FUNCTION_BLOCK FB_HybridStarter EXTENDS FB_BaseDevice
VAR_INPUT
	// The control output to the starter
    ControlOutput    AT %Q* : UINT;
	// The 5in1 state data word from the starter
    StatusInput      AT %I* : UINT;
	// The Max. current ampere word from the starter, in 10s of mA
    CurrentMaxInput  AT %I* : UINT;
	// The Thermal load input word from the starter
    ThermalLoadInput AT %I* : UINT;

    // Local copy of main control word as UINT (same as ControlOutput)
    uControl : UINT;
    // Local copy of main control word, individual bits that are translated to send to output
    stControl : ST_HybridStarterControlOutputBits;

    // Local copy of main status word as UINT (same as StatusInput)
    uStatus : UINT;
    // Local copy of main status word, translated to be readable as individual bits
    stStatus : ST_HybridStarterControlInputBits;

    // Max current word, multiplied by 10x, from tens of mA (same as CurrentMaxInput) to hundreds of mA, to be human readable
    uCurrentMilliamps : UINT;

    // Motor thermal load percentage (same as ThermalLoadInput)
    uThermalLoadPercent : UINT;
END_VAR

VAR
    uControlOutput : U_HybridStarterControlOutput;
    uControlInput1 : U_HybridStarterControlInput;
END_VAR

METHOD ReadControlInputs : BOOL
uStatus             := StatusInput;
uCurrentMilliamps   := CurrentMaxInput * 10; // Turn the 10s of mA value into 100s of mA
uThermalLoadPercent := ThermalLoadInput;

// Run the main input UINT through the union and store the bits in the local struct VAR
uControlInput1.uUint := uStatus;
stStatus             := uControlInput1.stBits;

ReadControlInputs := TRUE;
END_METHOD

METHOD RunForward : BOOL
VAR_INPUT
END_VAR
stControl.ForwardRunning := TRUE;
stControl.ReverseRunning := FALSE;
RunForward := TRUE;
END_METHOD

METHOD RunReverse : BOOL
VAR_INPUT
END_VAR
stControl.ForwardRunning := FALSE;
stControl.ReverseRunning := TRUE;
RunReverse := TRUE;
END_METHOD

METHOD SetNominalCurrent : BOOL
VAR_INPUT
	bit0 : BOOL;
	bit1 : BOOL;
	bit2 : BOOL;
	bit3 : BOOL;
END_VAR
stControl.NominalMotorCurrent0 := bit0;
stControl.NominalMotorCurrent1 := bit1;
stControl.NominalMotorCurrent2 := bit2;
stControl.NominalMotorCurrent3 := bit3;
stControl.IdentificationValid := TRUE;
SetNominalCurrent := TRUE;
END_METHOD

METHOD Stop : BOOL
VAR_INPUT
END_VAR
stControl.ForwardRunning := FALSE;
stControl.ReverseRunning := FALSE;

uControlOutput.stBits := stControl;
uControl := uControlOutput.uUint;
ControlOutput := uControl;

Stop := TRUE;
END_METHOD

METHOD WriteControlOutput : BOOL
VAR_INPUT
END_VAR
uControlOutput.stBits := stControl;
uControl := uControlOutput.uUint;
ControlOutput := uControl;
WriteControlOutput := TRUE;
END_METHOD

END_FUNCTION_BLOCK

(* stored: Version 1.1.0.1, ProductVersion 3.1.4024.12
   POU FB_HybridStarter: Id {40a43593-dd83-4697-9b52-2a55021f0aae}, SpecialFunc None
   Method ReadControlInputs: Id {032f4767-53a8-4f35-bf43-52c5c6b3764e}
   Method RunForward: Id {6b6c57d0-536f-4587-856c-f3044e21e237}
   Method RunReverse: Id {8e0f4a7c-2228-4fd1-b9f4-6c173716805d}
   Method SetNominalCurrent: Id {581c68a2-e07f-4d6e-bd1e-4df032e197e4}
   Method Stop: Id {4000f6dd-aedd-4472-ba4f-8472212352aa}
   Method WriteControlOutput: Id {bcdc0e86-075c-4243-9a30-bf472af78ee3} *)
